// TwinCAT 3 PLC project DALI_PLC
// ProgramVersion: 3.1.4024.0
// libraries:
//   Tc2_Standard, * (Beckhoff Automation GmbH)
//   Tc2_System, * (Beckhoff Automation GmbH)
//   Tc3_DALI, * (Beckhoff Automation GmbH)
//   Tc3_Module, * (Beckhoff Automation GmbH)
// project tree:
//   / DALI.TcTTO (not stored), PlcTask.TcTTO (not stored)
//   GVLs/ gvlDALI.TcGVL, gvlIO.TcGVL
//   POUs/ MAIN.TcPOU, POU_Comm.TcPOU (not stored), POU_DALIModule.TcPOU, POU_WALLLIGHT.TcPOU, PyADS_POU.TcPOU, POU_SWITCHES.TcPOU, POU_CURTAINS.TcPOU, POU_APPLIANCES.TcPOU, POU_SECURITY.TcPOU
// real-time tasks:
//   TASK PlcTask: cycle T#10ms, priority 10, ADS port 350
//   TASK DALI: cycle T#2ms, priority 4, ADS port 351
// I/O:
//   DEVICE Device 1 (Beckhoff CCAT)
//   DEVICE Device 2 (CX-BK)
//     Box 1 (CX-BK)
// variable links:
//   DALI_PLC/DALI_PLC Instance <-> Device 2 (CX-BK)/Box 1 (CX-BK)
//     DALI Inputs/gvlDALI.stKL6821InData/aData[{0..3}] <-> Term 3 (KL6821)/Channel 1/Data In {0..3}  (4 links)
//     DALI Inputs/gvlDALI.stKL6821InData/nStatus <-> Term 3 (KL6821)/Channel 1/State
//     DALI Outputs/gvlDALI.stKL6821OutData/aData[{0..3}] <-> Term 3 (KL6821)/Channel 1/Data Out {0..3}  (4 links)
//     DALI Outputs/gvlDALI.stKL6821OutData/nCtrl <-> Term 3 (KL6821)/Channel 1/Ctrl
//     PlcTask Inputs/gvlDALI.gButtonLightOn <-> Term 2 (KL1408)/Channel 1/Input
//     PlcTask Inputs/gvlDALI.gMotionLightOn <-> Term 2 (KL1408)/Channel 3/Input

// ---- GVLs/gvlDALI.TcGVL
{attribute 'qualified_only'}
(*
  gvlDALI — DALI dimmer bus, wall relay lights, and BTicino switch inputs.

  Standard array sizes (consistent across ALL apartments):
    DALI channels  : 1..16
    Wall relays    : 1..16  (physical links only wired for channels in use)
    Switch inputs  : 1..48  (3 × KL1809 16-channel terminals)
*)
VAR_GLOBAL

    // ── KL6821 DALI master terminal ──────────────────────────────────────────
    stKL6821InData      AT %I* : ST_KL6821InData;
    stKL6821OutData     AT %Q* : ST_KL6821OutData;

    // ── DALI dimmer levels (16 channels) ─────────────────────────────────────
    // Python writes aPyLevel[N] + rising edge on aPySetLevel[N] to dim.
    // PLC writes aPyActualLevel[N] as confirmed readback.
    aPyLevel            : ARRAY[1..16] OF BYTE;   // 0-254, desired level
    aPySetLevel         : ARRAY[1..16] OF BOOL;   // rising edge commits level
    aPyActualLevel      : ARRAY[1..16] OF BYTE;   // actual level → Python

    // ── Wall relay lights ────────────────────────────────────────────────────
    // aWallRelay[] are regular variables linked to relay output terminals in
    // the TwinCAT I/O tree (not AT %Q* auto-mapped).
    // Array sized to 16 so the same driver works for all apartments.
    aWallRelay          : ARRAY[1..16] OF BOOL;   // physical relay outputs (linked)
    aPyWallRelay        : ARRAY[1..16] OF BOOL;   // Python → PLC command
    aPyWallRelayState   : ARRAY[1..16] OF BOOL;   // PLC → Python readback

    // ── BTicino L4036 push-button inputs (KL1809 × 3 = 48 channels) ─────────
    aSwitch             : ARRAY[1..48] OF BOOL AT %I*;
    aPySwitchState      : ARRAY[1..48] OF BOOL;   // mirrored → Python readback

    // ── Legacy single-switch placeholder (kept for backwards compat) ─────────
    bSwitchOn           AT %I* : BOOL;
    gLightOn            : BOOL;
    gButtonLightOn      AT %I* : BOOL;
    gMotionLightOn      AT %I* : BOOL;

END_VAR

// ---- GVLs/gvlIO.TcGVL
{attribute 'qualified_only'}
(*
  gvlIO — Physical I/O and PyADS interface for all non-DALI devices.

  Naming convention (consistent across ALL apartments so the same Python
  driver works without changes; only _DEFAULT_* config dicts change):

    AT %I* vars   → auto-mapped to EtherCAT digital input terminals in
                    declaration order: KL1819 sensors come after KL1809 switches.
    Output vars   → no AT %Q*; link manually in TwinCAT I/O tree to the
                    relevant output terminal channels.
    aPy*Cmd[]     → Python writes these to command the PLC.
    aPy*State[]   → PLC writes these; Python polls them for readback.

  Standard array sizes for all apartments:
    Curtain motors : 1..16  (most apartments will use ≤ 8)
    Door sensors   : 1..16
    Window sensors : 1..16
    Motion sensors : 1..8
    Wall relays    : handled in gvlDALI (see there)
*)
VAR_GLOBAL

    // ═══════════════════════════════════════════════════════════════════════
    //  PHYSICAL INPUTS  (AT %I*)
    //  Terminal order after KL6821 + KL1809×3 (switches):
    //    Slots 1-2 → KL1819 × 2 → door sensors aDoorSensor[1..16]
    //    Slot  3   → KL1819      → window sensors aWindowSensor[1..8]  (8 ch)
    //    Slot  4   → KL1819      → window sensors aWindowSensor[9..16] + aMotionSensor[1..4]
    //    Slot  5   → KL1819 / KL1408 → bKeySwitch + spare
    // ═══════════════════════════════════════════════════════════════════════

    // Door magnetic sensors — TRUE = door open
    aDoorSensor     : ARRAY[1..16] OF BOOL AT %I*;

    // Window magnetic sensors — TRUE = window open
    aWindowSensor   : ARRAY[1..16] OF BOOL AT %I*;

    // PIR / motion sensors — TRUE = motion detected
    aMotionSensor   : ARRAY[1..8] OF BOOL AT %I*;

    // Key-based alarm/lockdown switch — TRUE = armed position
    bKeySwitch      : BOOL AT %I*;


    // ═══════════════════════════════════════════════════════════════════════
    //  PHYSICAL OUTPUTS  (linked manually in TwinCAT I/O tree)
    //  Curtain motors: 2 outputs per motor (Up / Down) → KL2xxx relay terms.
    //  Appliances:     1 output each                   → KL2xxx relay terms.
    // ═══════════════════════════════════════════════════════════════════════

    // Curtain motor directions (up to 16 motors, 2 signals each)
    aCurtainUp      : ARRAY[1..16] OF BOOL;   // HIGH = raise
    aCurtainDown    : ARRAY[1..16] OF BOOL;   // HIGH = lower

    // Appliance power relays
    bFridgeOut         : BOOL;
    bCoffeeMachineOut  : BOOL;
    bMicrowaveOut      : BOOL;


    // ═══════════════════════════════════════════════════════════════════════
    //  PyADS WRITE INTERFACE  — Python writes these to command the PLC
    // ═══════════════════════════════════════════════════════════════════════

    // Curtain command per motor: 0 = stop, 1 = up, 2 = down
    aPyCurtainCmd       : ARRAY[1..16] OF BYTE;

    // Physical-button curtain override (written by POU_SWITCHES; 0 = no press)
    // POU_CURTAINS gives this priority over the app command.
    aPyCurtainBtnCmd    : ARRAY[1..16] OF BYTE;

    // Appliance on/off commands
    bPyFridgeCmd        : BOOL;
    bPyCoffeeMachineCmd : BOOL;
    bPyMicrowaveCmd     : BOOL;

    // Security commands
    bPyAlarmArm         : BOOL;   // TRUE = arm alarm from app
    bPyLockdown         : BOOL;   // TRUE = activate house lockdown from app


    // ═══════════════════════════════════════════════════════════════════════
    //  PyADS READ INTERFACE  — PLC writes these; Python polls them
    // ═══════════════════════════════════════════════════════════════════════

    // Curtain motion state: 0 = stopped, 1 = moving up, 2 = moving down
    aPyCurtainState     : ARRAY[1..16] OF BYTE;

    // Appliance actual states
    bPyFridgeState         : BOOL;
    bPyCoffeeMachineState  : BOOL;
    bPyMicrowaveState      : BOOL;

    // Sensor readback (mirrored from physical inputs each PLC cycle)
    aPyDoorSensor       : ARRAY[1..16] OF BOOL;
    aPyWindowSensor     : ARRAY[1..16] OF BOOL;
    aPyMotionSensor     : ARRAY[1..8]  OF BOOL;
    bPyKeySwitch        : BOOL;

    // Security / alarm state
    bPyAlarmState       : BOOL;   // TRUE = alarm is currently armed
    bPyLockdownState    : BOOL;   // TRUE = lockdown is active
    bPyAlarmTriggered   : BOOL;   // TRUE = intrusion detected while armed

    // Shared lockdown flag — read by POU_DALIModule + POU_WALLLIGHT + POU_CURTAINS
    bLockdownActive     : BOOL;

END_VAR

// ---- POUs/POU_SWITCHES.TcPOU
(*
  POU_SWITCHES — BTicino L4036 push-button logic.

  Physical button mapping for Apartment 16
  ─────────────────────────────────────────
  Switches 1-6   → DALI room toggles  (bSwitch input on each FB_DALI102Dimmer*,
                   assigned directly in POU_DALIModule — no extra logic here)

  Switches 7-11  → Wall relay toggles  (edge-triggered: press = flip relay state)
    SW 7  → Wall Light 1  (aPyWallRelay[1])
    SW 8  → Wall Light 2  (aPyWallRelay[2])
    SW 9  → Wall Light 3  (aPyWallRelay[3])
    SW 10 → Wall Light 4  (aPyWallRelay[4])
    SW 11 → Wall Light 5  (aPyWallRelay[5])

  Switches 12-43 → Curtain hold-to-run  (level: hold = run, release = stop)
    SW 12/13 → Curtain 1 Up/Down
    SW 14/15 → Curtain 2 Up/Down
    SW 16/17 → Curtain 3 Up/Down
    SW 18/19 → Curtain 4 Up/Down
    SW 20/21 → Curtain 5 Up/Down
    SW 22/23 → Curtain 6 Up/Down
    SW 24/25 → Curtain 7 Up/Down
    SW 26/27 → Curtain 8 Up/Down

  Switches 28-48 → spare / future use

  Button commands for curtains are written to gvlIO.aPyCurtainBtnCmd[].
  POU_CURTAINS gives these priority over the app command.

  Switch states are mirrored to gvlDALI.aPySwitchState[] every cycle so
  Python can display the live button state in the app.
*)
PROGRAM POU_SWITCHES
VAR
    // Rising-edge detectors for wall relay toggles (one per relay, 1-indexed)
    artRelay    : ARRAY[1..16] OF R_TRIG;
    i           : INT;
END_VAR

// ── Mirror all switch states → Python readback ──────────────────────────────
FOR i := 1 TO 48 DO
    gvlDALI.aPySwitchState[i] := gvlDALI.aSwitch[i];
END_FOR

// ── Wall relay toggles (switches 7-11 → relays 1-5) ─────────────────────────
// artRelay[1] watches aSwitch[7], artRelay[2] watches aSwitch[8], etc.
FOR i := 1 TO 5 DO
    artRelay[i](CLK := gvlDALI.aSwitch[6 + i]);
    IF artRelay[i].Q THEN
        gvlDALI.aPyWallRelay[i] := NOT gvlDALI.aPyWallRelay[i];
    END_IF
END_FOR

// ── Curtain hold-to-run (switches 12-27 → motors 1-8) ───────────────────────
// Up   = switch 10 + (motor * 2)    → 12, 14, 16, 18, 20, 22, 24, 26
// Down = switch 10 + (motor * 2) + 1 → 13, 15, 17, 19, 21, 23, 25, 27
// A held button writes a non-zero cmd; releasing writes 0 (stop).
// POU_CURTAINS combines this with the app command.
FOR i := 1 TO 8 DO
    IF gvlDALI.aSwitch[10 + (i * 2)] THEN
        gvlIO.aPyCurtainBtnCmd[i] := 1;     // up
    ELSIF gvlDALI.aSwitch[10 + (i * 2) + 1] THEN
        gvlIO.aPyCurtainBtnCmd[i] := 2;     // down
    ELSE
        gvlIO.aPyCurtainBtnCmd[i] := 0;     // no button pressed
    END_IF
END_FOR

END_PROGRAM

// ---- POUs/POU_CURTAINS.TcPOU
(*
  POU_CURTAINS — Curtain motor control (up to 16 motors).

  Command priority (highest first):
    1. Lockdown active       → all motors driven DOWN (close curtains)
    2. Physical button press → aPyCurtainBtnCmd[i] (set by POU_SWITCHES)
    3. App command           → aPyCurtainCmd[i] (written by Python via PyADS)

  Commands:  0 = stop,  1 = up (raise),  2 = down (lower)

  Safety interlock: both Up and Down outputs for the same motor are NEVER
  set simultaneously.  Down is cleared before Up is set and vice-versa with
  a one-cycle gap enforced by the priority logic below.

  Physical outputs aCurtainUp[] / aCurtainDown[] are regular variables that
  must be linked to the motor relay output terminals in TwinCAT I/O tree.
*)
PROGRAM POU_CURTAINS
VAR
    i           : INT;
    nCmd        : BYTE;   // resolved command for current motor
END_VAR

FOR i := 1 TO 16 DO

    // ── Resolve effective command ────────────────────────────────────────────
    IF gvlIO.bLockdownActive THEN
        nCmd := 2;                              // lockdown → close all
    ELSIF gvlIO.aPyCurtainBtnCmd[i] <> 0 THEN
        nCmd := gvlIO.aPyCurtainBtnCmd[i];      // physical button has priority
    ELSE
        nCmd := gvlIO.aPyCurtainCmd[i];         // app command
    END_IF

    // ── Safety interlock + drive outputs ────────────────────────────────────
    CASE nCmd OF
        1:  // UP — clear Down first to avoid both-on glitch
            gvlIO.aCurtainDown[i] := FALSE;
            gvlIO.aCurtainUp[i]   := TRUE;
            gvlIO.aPyCurtainState[i] := 1;

        2:  // DOWN — clear Up first
            gvlIO.aCurtainUp[i]   := FALSE;
            gvlIO.aCurtainDown[i] := TRUE;
            gvlIO.aPyCurtainState[i] := 2;

        ELSE  // STOP (0 or any unknown value)
            gvlIO.aCurtainUp[i]   := FALSE;
            gvlIO.aCurtainDown[i] := FALSE;
            gvlIO.aPyCurtainState[i] := 0;
    END_CASE

END_FOR

END_PROGRAM

// ---- POUs/POU_DALIModule.TcPOU
(*
  POU_DALIModule — 16 Tridonic DALI ballasts via KL6821.

  Physical button mapping (aSwitch index per room):
    SW 1 → Living Room  (ch 1-4)
    SW 2 → Dining Room  (ch 5-8)
    SW 3 → Bedroom 1    (ch 9-10)
    SW 4 → Bedroom 2    (ch 11-12)
    SW 5 → Kitchen      (ch 13-14)
    SW 6 → Hallway      (ch 15-16)

  Lockdown: bOff := gvlIO.bLockdownActive on every FB call.
  Beckhoff's FB_DALI102Dimmer1Switch detects the rising edge internally,
  so setting bOff to TRUE fires a single DALI "Off" command (no bus spam).
*)
PROGRAM POU_DALIModule
VAR
    fbDALI102Dimmer1Switch      : FB_DALI102Dimmer1Switch(POU_Comm.fbKL6821Communication);
    fbDALI102Dimmer2Switch      : FB_DALI102Dimmer1Switch(POU_Comm.fbKL6821Communication);
    fbDALI102Dimmer3Switch      : FB_DALI102Dimmer1Switch(POU_Comm.fbKL6821Communication);
    fbDALI102Dimmer4Switch      : FB_DALI102Dimmer1Switch(POU_Comm.fbKL6821Communication);
    fbDALI102Dimmer5Switch      : FB_DALI102Dimmer1Switch(POU_Comm.fbKL6821Communication);
    fbDALI102Dimmer6Switch      : FB_DALI102Dimmer1Switch(POU_Comm.fbKL6821Communication);
    fbDALI102Dimmer7Switch      : FB_DALI102Dimmer1Switch(POU_Comm.fbKL6821Communication);
    fbDALI102Dimmer8Switch      : FB_DALI102Dimmer1Switch(POU_Comm.fbKL6821Communication);
    fbDALI102Dimmer9Switch      : FB_DALI102Dimmer1Switch(POU_Comm.fbKL6821Communication);
    fbDALI102Dimmer10Switch     : FB_DALI102Dimmer1Switch(POU_Comm.fbKL6821Communication);
    fbDALI102Dimmer11Switch     : FB_DALI102Dimmer1Switch(POU_Comm.fbKL6821Communication);
    fbDALI102Dimmer12Switch     : FB_DALI102Dimmer1Switch(POU_Comm.fbKL6821Communication);
    fbDALI102Dimmer13Switch     : FB_DALI102Dimmer1Switch(POU_Comm.fbKL6821Communication);
    fbDALI102Dimmer14Switch     : FB_DALI102Dimmer1Switch(POU_Comm.fbKL6821Communication);
    fbDALI102Dimmer15Switch     : FB_DALI102Dimmer1Switch(POU_Comm.fbKL6821Communication);
    fbDALI102Dimmer16Switch     : FB_DALI102Dimmer1Switch(POU_Comm.fbKL6821Communication);

    bInitialize                 : BOOL := FALSE;

    // Per-dimmer local variables (level, setlevel trigger, actual readback)
    bSetLevel_1   : BOOL;  nLevel_1   : BYTE := 254;  nActualLevel_1   : BYTE;
    bSetLevel_2   : BOOL;  nLevel_2   : BYTE := 254;  nActualLevel_2   : BYTE;
    bSetLevel_3   : BOOL;  nLevel_3   : BYTE := 254;  nActualLevel_3   : BYTE;
    bSetLevel_4   : BOOL;  nLevel_4   : BYTE := 254;  nActualLevel_4   : BYTE;
    bSetLevel_5   : BOOL;  nLevel_5   : BYTE := 254;  nActualLevel_5   : BYTE;
    bSetLevel_6   : BOOL;  nLevel_6   : BYTE := 254;  nActualLevel_6   : BYTE;
    bSetLevel_7   : BOOL;  nLevel_7   : BYTE := 254;  nActualLevel_7   : BYTE;
    bSetLevel_8   : BOOL;  nLevel_8   : BYTE := 254;  nActualLevel_8   : BYTE;
    bSetLevel_9   : BOOL;  nLevel_9   : BYTE := 254;  nActualLevel_9   : BYTE;
    bSetLevel_10  : BOOL;  nLevel_10  : BYTE := 254;  nActualLevel_10  : BYTE;
    bSetLevel_11  : BOOL;  nLevel_11  : BYTE := 254;  nActualLevel_11  : BYTE;
    bSetLevel_12  : BOOL;  nLevel_12  : BYTE := 254;  nActualLevel_12  : BYTE;
    bSetLevel_13  : BOOL;  nLevel_13  : BYTE := 254;  nActualLevel_13  : BYTE;
    bSetLevel_14  : BOOL;  nLevel_14  : BYTE := 254;  nActualLevel_14  : BYTE;
    bSetLevel_15  : BOOL;  nLevel_15  : BYTE := 254;  nActualLevel_15  : BYTE;
    bSetLevel_16  : BOOL;  nLevel_16  : BYTE := 254;  nActualLevel_16  : BYTE;

    // Common options (shared across all dimmers)
    nLevelMemoryMode    : BYTE  := 70;
    tCycleActualLevel   : TIME  := T#5S;
    nOptions            : DWORD := 0;
END_VAR

// ── Sync PyADS inputs → per-dimmer variables ────────────────────────────────
bSetLevel_1  := gvlDALI.aPySetLevel[1];   nLevel_1  := gvlDALI.aPyLevel[1];
bSetLevel_2  := gvlDALI.aPySetLevel[2];   nLevel_2  := gvlDALI.aPyLevel[2];
bSetLevel_3  := gvlDALI.aPySetLevel[3];   nLevel_3  := gvlDALI.aPyLevel[3];
bSetLevel_4  := gvlDALI.aPySetLevel[4];   nLevel_4  := gvlDALI.aPyLevel[4];
bSetLevel_5  := gvlDALI.aPySetLevel[5];   nLevel_5  := gvlDALI.aPyLevel[5];
bSetLevel_6  := gvlDALI.aPySetLevel[6];   nLevel_6  := gvlDALI.aPyLevel[6];
bSetLevel_7  := gvlDALI.aPySetLevel[7];   nLevel_7  := gvlDALI.aPyLevel[7];
bSetLevel_8  := gvlDALI.aPySetLevel[8];   nLevel_8  := gvlDALI.aPyLevel[8];
bSetLevel_9  := gvlDALI.aPySetLevel[9];   nLevel_9  := gvlDALI.aPyLevel[9];
bSetLevel_10 := gvlDALI.aPySetLevel[10];  nLevel_10 := gvlDALI.aPyLevel[10];
bSetLevel_11 := gvlDALI.aPySetLevel[11];  nLevel_11 := gvlDALI.aPyLevel[11];
bSetLevel_12 := gvlDALI.aPySetLevel[12];  nLevel_12 := gvlDALI.aPyLevel[12];
bSetLevel_13 := gvlDALI.aPySetLevel[13];  nLevel_13 := gvlDALI.aPyLevel[13];
bSetLevel_14 := gvlDALI.aPySetLevel[14];  nLevel_14 := gvlDALI.aPyLevel[14];
bSetLevel_15 := gvlDALI.aPySetLevel[15];  nLevel_15 := gvlDALI.aPyLevel[15];
bSetLevel_16 := gvlDALI.aPySetLevel[16];  nLevel_16 := gvlDALI.aPyLevel[16];

// ── Dimmer 1 — Living Room (SW 1) ────────────────────────────────────────────
fbDALI102Dimmer1Switch(
    bInitialize          := bInitialize,
    nAddress             := 1,
    eAddressType         := E_DALIAddressType.Short,
    bSwitch              := gvlDALI.aSwitch[1],
    bOff                 := gvlIO.bLockdownActive,
    bSetLevel            := bSetLevel_1,
    nLevel               := nLevel_1,
    nLevelMemoryMode     := nLevelMemoryMode,
    tCycleActualLevel    := tCycleActualLevel,
    nOptions             := nOptions
);
nActualLevel_1 := fbDALI102Dimmer1Switch.nActualLevel;
gvlDALI.aPyActualLevel[1] := nActualLevel_1;

// ── Dimmer 2 — Living Room (SW 1) ────────────────────────────────────────────
fbDALI102Dimmer2Switch(
    bInitialize          := bInitialize,
    nAddress             := 2,
    eAddressType         := E_DALIAddressType.Short,
    bSwitch              := gvlDALI.aSwitch[1],
    bOff                 := gvlIO.bLockdownActive,
    bSetLevel            := bSetLevel_2,
    nLevel               := nLevel_2,
    nLevelMemoryMode     := nLevelMemoryMode,
    tCycleActualLevel    := tCycleActualLevel,
    nOptions             := nOptions
);
nActualLevel_2 := fbDALI102Dimmer2Switch.nActualLevel;
gvlDALI.aPyActualLevel[2] := nActualLevel_2;

// ── Dimmer 3 — Living Room (SW 1) ────────────────────────────────────────────
fbDALI102Dimmer3Switch(
    bInitialize          := bInitialize,
    nAddress             := 3,
    eAddressType         := E_DALIAddressType.Short,
    bSwitch              := gvlDALI.aSwitch[1],
    bOff                 := gvlIO.bLockdownActive,
    bSetLevel            := bSetLevel_3,
    nLevel               := nLevel_3,
    nLevelMemoryMode     := nLevelMemoryMode,
    tCycleActualLevel    := tCycleActualLevel,
    nOptions             := nOptions
);
nActualLevel_3 := fbDALI102Dimmer3Switch.nActualLevel;
gvlDALI.aPyActualLevel[3] := nActualLevel_3;

// ── Dimmer 4 — Living Room (SW 1) ────────────────────────────────────────────
fbDALI102Dimmer4Switch(
    bInitialize          := bInitialize,
    nAddress             := 4,
    eAddressType         := E_DALIAddressType.Short,
    bSwitch              := gvlDALI.aSwitch[1],
    bOff                 := gvlIO.bLockdownActive,
    bSetLevel            := bSetLevel_4,
    nLevel               := nLevel_4,
    nLevelMemoryMode     := nLevelMemoryMode,
    tCycleActualLevel    := tCycleActualLevel,
    nOptions             := nOptions
);
nActualLevel_4 := fbDALI102Dimmer4Switch.nActualLevel;
gvlDALI.aPyActualLevel[4] := nActualLevel_4;

// ── Dimmer 5 — Dining Room (SW 2) ────────────────────────────────────────────
fbDALI102Dimmer5Switch(
    bInitialize          := bInitialize,
    nAddress             := 5,
    eAddressType         := E_DALIAddressType.Short,
    bSwitch              := gvlDALI.aSwitch[2],
    bOff                 := gvlIO.bLockdownActive,
    bSetLevel            := bSetLevel_5,
    nLevel               := nLevel_5,
    nLevelMemoryMode     := nLevelMemoryMode,
    tCycleActualLevel    := tCycleActualLevel,
    nOptions             := nOptions
);
nActualLevel_5 := fbDALI102Dimmer5Switch.nActualLevel;
gvlDALI.aPyActualLevel[5] := nActualLevel_5;

// ── Dimmer 6 — Dining Room (SW 2) ────────────────────────────────────────────
fbDALI102Dimmer6Switch(
    bInitialize          := bInitialize,
    nAddress             := 6,
    eAddressType         := E_DALIAddressType.Short,
    bSwitch              := gvlDALI.aSwitch[2],
    bOff                 := gvlIO.bLockdownActive,
    bSetLevel            := bSetLevel_6,
    nLevel               := nLevel_6,
    nLevelMemoryMode     := nLevelMemoryMode,
    tCycleActualLevel    := tCycleActualLevel,
    nOptions             := nOptions
);
nActualLevel_6 := fbDALI102Dimmer6Switch.nActualLevel;
gvlDALI.aPyActualLevel[6] := nActualLevel_6;

// ── Dimmer 7 — Dining Room (SW 2) ────────────────────────────────────────────
fbDALI102Dimmer7Switch(
    bInitialize          := bInitialize,
    nAddress             := 7,
    eAddressType         := E_DALIAddressType.Short,
    bSwitch              := gvlDALI.aSwitch[2],
    bOff                 := gvlIO.bLockdownActive,
    bSetLevel            := bSetLevel_7,
    nLevel               := nLevel_7,
    nLevelMemoryMode     := nLevelMemoryMode,
    tCycleActualLevel    := tCycleActualLevel,
    nOptions             := nOptions
);
nActualLevel_7 := fbDALI102Dimmer7Switch.nActualLevel;
gvlDALI.aPyActualLevel[7] := nActualLevel_7;

// ── Dimmer 8 — Dining Room (SW 2) ────────────────────────────────────────────
fbDALI102Dimmer8Switch(
    bInitialize          := bInitialize,
    nAddress             := 8,
    eAddressType         := E_DALIAddressType.Short,
    bSwitch              := gvlDALI.aSwitch[2],
    bOff                 := gvlIO.bLockdownActive,
    bSetLevel            := bSetLevel_8,
    nLevel               := nLevel_8,
    nLevelMemoryMode     := nLevelMemoryMode,
    tCycleActualLevel    := tCycleActualLevel,
    nOptions             := nOptions
);
nActualLevel_8 := fbDALI102Dimmer8Switch.nActualLevel;
gvlDALI.aPyActualLevel[8] := nActualLevel_8;

// ── Dimmer 9 — Bedroom 1 (SW 3) ──────────────────────────────────────────────
fbDALI102Dimmer9Switch(
    bInitialize          := bInitialize,
    nAddress             := 9,
    eAddressType         := E_DALIAddressType.Short,
    bSwitch              := gvlDALI.aSwitch[3],
    bOff                 := gvlIO.bLockdownActive,
    bSetLevel            := bSetLevel_9,
    nLevel               := nLevel_9,
    nLevelMemoryMode     := nLevelMemoryMode,
    tCycleActualLevel    := tCycleActualLevel,
    nOptions             := nOptions
);
nActualLevel_9 := fbDALI102Dimmer9Switch.nActualLevel;
gvlDALI.aPyActualLevel[9] := nActualLevel_9;

// ── Dimmer 10 — Bedroom 1 (SW 3) ─────────────────────────────────────────────
fbDALI102Dimmer10Switch(
    bInitialize          := bInitialize,
    nAddress             := 10,
    eAddressType         := E_DALIAddressType.Short,
    bSwitch              := gvlDALI.aSwitch[3],
    bOff                 := gvlIO.bLockdownActive,
    bSetLevel            := bSetLevel_10,
    nLevel               := nLevel_10,
    nLevelMemoryMode     := nLevelMemoryMode,
    tCycleActualLevel    := tCycleActualLevel,
    nOptions             := nOptions
);
nActualLevel_10 := fbDALI102Dimmer10Switch.nActualLevel;
gvlDALI.aPyActualLevel[10] := nActualLevel_10;

// ── Dimmer 11 — Bedroom 2 (SW 4) ─────────────────────────────────────────────
fbDALI102Dimmer11Switch(
    bInitialize          := bInitialize,
    nAddress             := 11,
    eAddressType         := E_DALIAddressType.Short,
    bSwitch              := gvlDALI.aSwitch[4],
    bOff                 := gvlIO.bLockdownActive,
    bSetLevel            := bSetLevel_11,
    nLevel               := nLevel_11,
    nLevelMemoryMode     := nLevelMemoryMode,
    tCycleActualLevel    := tCycleActualLevel,
    nOptions             := nOptions
);
nActualLevel_11 := fbDALI102Dimmer11Switch.nActualLevel;
gvlDALI.aPyActualLevel[11] := nActualLevel_11;

// ── Dimmer 12 — Bedroom 2 (SW 4) ─────────────────────────────────────────────
fbDALI102Dimmer12Switch(
    bInitialize          := bInitialize,
    nAddress             := 12,
    eAddressType         := E_DALIAddressType.Short,
    bSwitch              := gvlDALI.aSwitch[4],
    bOff                 := gvlIO.bLockdownActive,
    bSetLevel            := bSetLevel_12,
    nLevel               := nLevel_12,
    nLevelMemoryMode     := nLevelMemoryMode,
    tCycleActualLevel    := tCycleActualLevel,
    nOptions             := nOptions
);
nActualLevel_12 := fbDALI102Dimmer12Switch.nActualLevel;
gvlDALI.aPyActualLevel[12] := nActualLevel_12;

// ── Dimmer 13 — Kitchen (SW 5) ───────────────────────────────────────────────
fbDALI102Dimmer13Switch(
    bInitialize          := bInitialize,
    nAddress             := 13,
    eAddressType         := E_DALIAddressType.Short,
    bSwitch              := gvlDALI.aSwitch[5],
    bOff                 := gvlIO.bLockdownActive,
    bSetLevel            := bSetLevel_13,
    nLevel               := nLevel_13,
    nLevelMemoryMode     := nLevelMemoryMode,
    tCycleActualLevel    := tCycleActualLevel,
    nOptions             := nOptions
);
nActualLevel_13 := fbDALI102Dimmer13Switch.nActualLevel;
gvlDALI.aPyActualLevel[13] := nActualLevel_13;

// ── Dimmer 14 — Kitchen (SW 5) ───────────────────────────────────────────────
fbDALI102Dimmer14Switch(
    bInitialize          := bInitialize,
    nAddress             := 14,
    eAddressType         := E_DALIAddressType.Short,
    bSwitch              := gvlDALI.aSwitch[5],
    bOff                 := gvlIO.bLockdownActive,
    bSetLevel            := bSetLevel_14,
    nLevel               := nLevel_14,
    nLevelMemoryMode     := nLevelMemoryMode,
    tCycleActualLevel    := tCycleActualLevel,
    nOptions             := nOptions
);
nActualLevel_14 := fbDALI102Dimmer14Switch.nActualLevel;
gvlDALI.aPyActualLevel[14] := nActualLevel_14;

// ── Dimmer 15 — Hallway (SW 6) ───────────────────────────────────────────────
fbDALI102Dimmer15Switch(
    bInitialize          := bInitialize,
    nAddress             := 15,
    eAddressType         := E_DALIAddressType.Short,
    bSwitch              := gvlDALI.aSwitch[6],
    bOff                 := gvlIO.bLockdownActive,
    bSetLevel            := bSetLevel_15,
    nLevel               := nLevel_15,
    nLevelMemoryMode     := nLevelMemoryMode,
    tCycleActualLevel    := tCycleActualLevel,
    nOptions             := nOptions
);
nActualLevel_15 := fbDALI102Dimmer15Switch.nActualLevel;
gvlDALI.aPyActualLevel[15] := nActualLevel_15;

// ── Dimmer 16 — Hallway (SW 6) ───────────────────────────────────────────────
fbDALI102Dimmer16Switch(
    bInitialize          := bInitialize,
    nAddress             := 16,
    eAddressType         := E_DALIAddressType.Short,
    bSwitch              := gvlDALI.aSwitch[6],
    bOff                 := gvlIO.bLockdownActive,
    bSetLevel            := bSetLevel_16,
    nLevel               := nLevel_16,
    nLevelMemoryMode     := nLevelMemoryMode,
    tCycleActualLevel    := tCycleActualLevel,
    nOptions             := nOptions
);
nActualLevel_16 := fbDALI102Dimmer16Switch.nActualLevel;
gvlDALI.aPyActualLevel[16] := nActualLevel_16;

END_PROGRAM

// ---- POUs/POU_WALLLIGHT.TcPOU
(*
  POU_WALLLIGHT — Wall relay light control.

  Reads Python commands from gvlDALI.aPyWallRelay[] and drives
  gvlDALI.aWallRelay[] (linked to physical relay output terminals).

  Lockdown override: when gvlIO.bLockdownActive is TRUE all relays are
  forced off regardless of the app command.

  Array[1..16] covers all apartments; only wired channels have
  a physical relay linked in the I/O tree, so unused indices are harmless.
*)
PROGRAM POU_WALLLIGHT
VAR
    i : INT;
END_VAR

// ── Drive physical relay outputs ────────────────────────────────────────────
FOR i := 1 TO 16 DO
    IF gvlIO.bLockdownActive THEN
        // Lockdown: force all wall lights off
        gvlDALI.aWallRelay[i] := FALSE;
    ELSE
        // Normal: follow app command
        gvlDALI.aWallRelay[i] := gvlDALI.aPyWallRelay[i];
    END_IF
END_FOR

END_PROGRAM

// ---- POUs/MAIN.TcPOU
(*
  MAIN — Task entry point.  Execution order matters:

    1. POU_SECURITY   — evaluate sensors + set bLockdownActive first so all
                        other POUs can read the flag in the same cycle.
    2. POU_SWITCHES   — edge-detect BTicino buttons; write relay toggles and
                        curtain button commands.
    3. POU_DALIModule — drive 16 DALI dimmers (reads bLockdownActive).
    4. POU_WALLLIGHT  — drive relay lights (reads bLockdownActive).
    5. POU_CURTAINS   — drive curtain motors (reads bLockdownActive + btn cmds).
    6. POU_APPLIANCES — drive appliance relays (reads bLockdownActive).
    7. PyADS_POU      — mirror outputs → Python readback variables.
*)
PROGRAM MAIN
VAR
END_VAR

POU_SECURITY();     // 1 — sensors + lockdown flag
POU_SWITCHES();     // 2 — BTicino button logic
POU_DALIModule();   // 3 — DALI dimmers
POU_WALLLIGHT();    // 4 — relay wall lights
POU_CURTAINS();     // 5 — curtain motors
POU_APPLIANCES();   // 6 — smart appliances
PyADS_POU();        // 7 — readback mirror

END_PROGRAM

// ---- POUs/POU_SECURITY.TcPOU
(*
  POU_SECURITY — Alarm, lockdown, and sensor management.

  Alarm arming:
    Arm sources  : physical key switch (bKeySwitch) OR app command (bPyAlarmArm).
    Disarm       : both sources must be FALSE to disarm.
    Trigger      : any door/window open, or motion detected, while armed.
    Clear trigger: disarming automatically clears the triggered state.

  Lockdown mode:
    Activated by bPyLockdown (app command).
    Sets gvlIO.bLockdownActive which is read by:
      POU_WALLLIGHT  → forces all relay lights off
      POU_CURTAINS   → forces all curtains down (closed)
      POU_APPLIANCES → turns off heat appliances
      POU_DALIModule → fires DALI Off command once on activation

  Sensor readback:
    Physical inputs are mirrored to aPy* vars every PLC cycle so Python
    can display live states in the app without extra ADS reads.
*)
PROGRAM POU_SECURITY
VAR
    bAlarmArmed         : BOOL;
    bAlarmTriggered     : BOOL;
    bAnyIntrusion       : BOOL;
    i                   : INT;
END_VAR

// ── Sensor readback → Python ─────────────────────────────────────────────────
FOR i := 1 TO 16 DO
    gvlIO.aPyDoorSensor[i]   := gvlIO.aDoorSensor[i];
    gvlIO.aPyWindowSensor[i] := gvlIO.aWindowSensor[i];
END_FOR
FOR i := 1 TO 8 DO
    gvlIO.aPyMotionSensor[i] := gvlIO.aMotionSensor[i];
END_FOR
gvlIO.bPyKeySwitch := gvlIO.bKeySwitch;

// ── Alarm arm state ──────────────────────────────────────────────────────────
// Key switch (physical) OR app command arms the alarm.
// Both must be FALSE to disarm.
bAlarmArmed := gvlIO.bKeySwitch OR gvlIO.bPyAlarmArm;

// ── Intrusion detection ──────────────────────────────────────────────────────
bAnyIntrusion := FALSE;
IF bAlarmArmed THEN
    FOR i := 1 TO 16 DO
        IF gvlIO.aDoorSensor[i]   THEN bAnyIntrusion := TRUE; END_IF
        IF gvlIO.aWindowSensor[i] THEN bAnyIntrusion := TRUE; END_IF
    END_FOR
    FOR i := 1 TO 8 DO
        IF gvlIO.aMotionSensor[i] THEN bAnyIntrusion := TRUE; END_IF
    END_FOR
END_IF

// Latch trigger; clear only on disarm
IF bAnyIntrusion AND NOT bAlarmTriggered THEN
    bAlarmTriggered := TRUE;
END_IF
IF NOT bAlarmArmed THEN
    bAlarmTriggered := FALSE;
END_IF

// ── Lockdown activation ──────────────────────────────────────────────────────
// bLockdownActive is the shared flag consumed by all other POUs.
gvlIO.bLockdownActive := gvlIO.bPyLockdown;

// ── Security state readback → Python ────────────────────────────────────────
gvlIO.bPyAlarmState     := bAlarmArmed;
gvlIO.bPyAlarmTriggered := bAlarmTriggered;
gvlIO.bPyLockdownState  := gvlIO.bLockdownActive;

END_PROGRAM

// ---- POUs/POU_APPLIANCES.TcPOU
(*
  POU_APPLIANCES — Smart appliance relay control.

  Devices: fridge, coffee machine, microwave (expandable).
  Python writes bPy*Cmd; PLC drives physical relay output; state is mirrored
  back to bPy*State for Python readback.

  During lockdown the coffee machine and microwave are forced off (fridge
  stays on to protect food).

  Physical output variables (bFridgeOut, etc.) are regular variables that
  must be linked to relay output terminals in the TwinCAT I/O tree.
*)
PROGRAM POU_APPLIANCES
VAR
END_VAR

// ── Drive relay outputs ──────────────────────────────────────────────────────
IF gvlIO.bLockdownActive THEN
    // Lockdown: keep fridge running, turn off heat-producing appliances
    gvlIO.bFridgeOut        := gvlIO.bPyFridgeCmd;    // fridge stays as-is
    gvlIO.bCoffeeMachineOut := FALSE;
    gvlIO.bMicrowaveOut     := FALSE;
ELSE
    gvlIO.bFridgeOut        := gvlIO.bPyFridgeCmd;
    gvlIO.bCoffeeMachineOut := gvlIO.bPyCoffeeMachineCmd;
    gvlIO.bMicrowaveOut     := gvlIO.bPyMicrowaveCmd;
END_IF

// ── Readback → Python ────────────────────────────────────────────────────────
gvlIO.bPyFridgeState        := gvlIO.bFridgeOut;
gvlIO.bPyCoffeeMachineState := gvlIO.bCoffeeMachineOut;
gvlIO.bPyMicrowaveState     := gvlIO.bMicrowaveOut;

END_PROGRAM

// ---- POUs/PyADS_POU.TcPOU
(*
  PyADS_POU — Mirrors PLC outputs back to the PyADS read-interface variables.

  This POU is the "readback" layer: it copies physically-driven outputs into
  the aPy*State variables that Python reads via ADS.
  All actual sensor readbacks (door/window/motion) and security state are
  handled directly in POU_SECURITY; this POU covers DALI + relay + curtain
  + appliance where the "state" is derived from the output variable itself.
*)
PROGRAM PyADS_POU
VAR
    i : INT;
END_VAR

// ── Wall relay readback ───────────────────────────────────────────────────────
// Copy physical relay output (after lockdown override) back to Python readback.
FOR i := 1 TO 16 DO
    gvlDALI.aPyWallRelayState[i] := gvlDALI.aWallRelay[i];
END_FOR

// ── Switch state readback ─────────────────────────────────────────────────────
// Also done in POU_SWITCHES; kept here as belt-and-suspenders.
FOR i := 1 TO 48 DO
    gvlDALI.aPySwitchState[i] := gvlDALI.aSwitch[i];
END_FOR

// ── Curtain state readback ────────────────────────────────────────────────────
// aPyCurtainState[] is written by POU_CURTAINS — no duplication needed here.

// ── Appliance state readback ──────────────────────────────────────────────────
// bPy*State written by POU_APPLIANCES — no duplication needed here.

// ── Security / sensor readback ────────────────────────────────────────────────
// aPyDoorSensor[], aPyWindowSensor[], aPyMotionSensor[], bPyAlarmState, etc.
// are all written by POU_SECURITY — no duplication needed here.

END_PROGRAM
